// TIA Portal V20 export
// export: Created 2025-09-12T17:59:00.0000000Z, ExportSetting WithDefaults
FUNCTION_BLOCK "FB400_EM_Damper"   // FB, SCL
TITLE = EM-400: Damper Control
AUTHOR : Dallas Levine
VERSION : 0.1
// This block contains all logic for the Damper Equipment Module (EM-400).
// stored: AutoNumber true, IsRetain false
   VAR_INPUT
      Enable : Bool;   // Enables the block's execution.
   END_VAR
   VAR
      UDT : "UDT400_EM_Damper";   // The data interface for the Damper Equipment Module.
   END_VAR
BEGIN
   REGION Placeholder for SCL Code 

   END_REGION
END_FUNCTION_BLOCK
